PROGRAM G7_Palpage_Sommet_L
VAR_INPUT	SFCInit:BOOL;	END_VAR
VAR

	a1: LREAL;
	b1: LREAL;
	test_PalpSommet:BOOL;
END_VAR

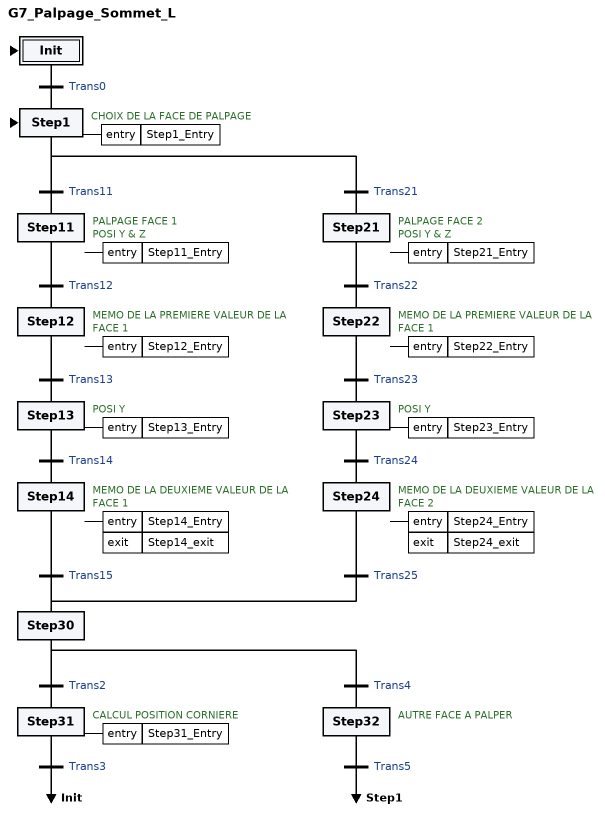
INITIAL_STEP Init:
END_STEP
TRANSITION FROM Init TO Step1
    := Trans0;
END_TRANSITION
// CHOIX DE LA FACE DE PALPAGE
STEP Step1:
    Step1_Entry(P1);  // entry action
END_STEP
TRANSITION FROM Step1 TO Step11
    := Trans11;
END_TRANSITION
// 																PALPAGE FACE 1
// POSI Y & Z
//
STEP Step11:
    Step11_Entry(P1);  // entry action
END_STEP
TRANSITION FROM Step11 TO Step12
    := Trans12;
END_TRANSITION
// MEMO DE LA PREMIERE VALEUR DE LA FACE 1
STEP Step12:
    Step12_Entry(P1);  // entry action
END_STEP
TRANSITION FROM Step12 TO Step13
    := Trans13;
END_TRANSITION
// POSI Y
STEP Step13:
    Step13_Entry(P1);  // entry action
END_STEP
TRANSITION FROM Step13 TO Step14
    := Trans14;
END_TRANSITION
// MEMO DE LA DEUXIEME VALEUR DE LA FACE 1
STEP Step14:
    Step14_Entry(P1);  // entry action
    Step14_exit(P0);  // exit action
END_STEP
TRANSITION FROM Step14 TO Step30
    := Trans15;
END_TRANSITION
TRANSITION FROM Step1 TO Step21
    := Trans21;
END_TRANSITION
// 																PALPAGE FACE 2
// POSI Y & Z
//
STEP Step21:
    Step21_Entry(P1);  // entry action
END_STEP
TRANSITION FROM Step21 TO Step22
    := Trans22;
END_TRANSITION
// MEMO DE LA PREMIERE VALEUR DE LA FACE 1
STEP Step22:
    Step22_Entry(P1);  // entry action
END_STEP
TRANSITION FROM Step22 TO Step23
    := Trans23;
END_TRANSITION
// POSI Y
STEP Step23:
    Step23_Entry(P1);  // entry action
END_STEP
TRANSITION FROM Step23 TO Step24
    := Trans24;
END_TRANSITION
// MEMO DE LA DEUXIEME VALEUR DE LA FACE 2
STEP Step24:
    Step24_Entry(P1);  // entry action
    Step24_exit(P0);  // exit action
END_STEP
TRANSITION FROM Step24 TO Step30
    := Trans25;
END_TRANSITION
STEP Step30:
END_STEP
TRANSITION FROM Step30 TO Step31
    := Trans2;
END_TRANSITION
TRANSITION FROM Step30 TO Step32
    := Trans4;
END_TRANSITION
// AUTRE FACE A PALPER
STEP Step32:
END_STEP
TRANSITION FROM Step32 TO Step1
    := Trans5;
END_TRANSITION
// 										CALCUL POSITION CORNIERE
//
//
STEP Step31:
    Step31_Entry(P1);  // entry action
END_STEP
TRANSITION FROM Step31 TO Init
    := Trans3;
END_TRANSITION

ACTION Step1_Entry:
CASE Face_Cible_Cycle OF	  
	1 : IF NOT Palpage_OK_Face_2 THEN
			Top_Palpage_Face_2 := TRUE;
			Top_Palpage_Face_1 := FALSE;
		ELSIF NOT Palpage_OK_Face_1 THEN
			Top_Palpage_Face_1 := TRUE;
			Top_Palpage_Face_2 := FALSE;
		ELSE
			Top_Palpage_Face_1 := FALSE;
			Top_Palpage_Face_2 := FALSE;
		END_IF;

	2,3 : 	IF NOT Palpage_OK_Face_1 THEN
			Top_Palpage_Face_1 := TRUE;
			Top_Palpage_Face_2 := FALSE;
		ELSIF NOT Palpage_OK_Face_2 THEN
			Top_Palpage_Face_2 := TRUE;
			Top_Palpage_Face_1 := FALSE;
		ELSE
			Top_Palpage_Face_1 := FALSE;
			Top_Palpage_Face_2 := FALSE;
		END_IF;
END_CASE;


IF Top_Palpage_Face_1 THEN
	 Face_Cible_Palpage := 1;
ELSIF  Top_Palpage_Face_2 THEN
	 Face_Cible_Palpage := 2;
ELSE
	Face_Cible_Palpage := 0;
END_IF;


IF Face_Cible_Palpage <> 0 THEN
	Face_Cible 		:= Face_Cible_Palpage;
	Face_En_Pos 	:= FALSE;
	Top_Face 		:= TRUE;
END_IF;
END_ACTION

ACTION Step11_Entry:
Pos_cible_Y_Laser := Offset_Y_Laser_REF + Hauteur_Aile - Ep_Ame - 5;
En_pos_Y_Laser :=FALSE;
Top_Y_Laser := TRUE;

Pos_cible_Z_Laser := Offset_Z_Laser_REF - Global_Divers.EP_Aile - 10;	//10 sécu arbitraire, à peut être adapter selon test
En_pos_Z_Laser :=FALSE;
Top_Z_Laser := TRUE;
END_ACTION

ACTION Step12_Entry:
Memo_Face_1_Y_1 := Hauteur_Aile - Ep_Ame - 5;
Memo_Face_1_Z_1 := Global_Divers.EP_Aile + Prog_Capacitance_Actual_Value_mm - 10;
END_ACTION

ACTION Step13_Entry:
Pos_cible_Y_Laser := Offset_Y_Laser_REF;
En_pos_Y_Laser :=FALSE;
Top_Y_Laser := TRUE;
END_ACTION

ACTION Step14_Entry:
Memo_Face_1_Y_2 := Ep_Ame;
Memo_Face_1_Z_2 := Global_Divers.EP_Aile + Prog_Capacitance_Actual_Value_mm - 10;
END_ACTION

ACTION Step14_exit:
Palpage_OK_Face_1:=true;
END_ACTION

ACTION Step21_Entry:
Pos_cible_Y_Laser := Offset_Y_Laser_OPP_REF - Largeur_Ame + Global_Divers.EP_Aile + 5;
En_pos_Y_Laser :=FALSE;
Top_Y_Laser := TRUE;

Pos_cible_Z_Laser := Offset_Z_Laser_OPP_REF - Ep_Ame - 10;
En_pos_Z_Laser :=FALSE;
Top_Z_Laser := TRUE;
END_ACTION

ACTION Step22_Entry:
Memo_Face_2_Y_1 := Largeur_Ame - Global_Divers.EP_Aile - 5;
Memo_Face_2_Z_1 := Ep_Ame + Prog_Capacitance_Actual_Value_mm - 10;
END_ACTION

ACTION Step23_Entry:
Pos_cible_Y_Laser := Offset_Y_Laser_OPP_REF;
En_pos_Y_Laser :=FALSE;
Top_Y_Laser := TRUE;
END_ACTION

ACTION Step24_Entry:
Memo_Face_2_Y_1 := Global_Divers.EP_Aile;
Memo_Face_2_Z_1 := Ep_Ame + Prog_Capacitance_Actual_Value_mm - 10;
END_ACTION

ACTION Step24_exit:
Palpage_OK_Face_2:=true;
END_ACTION

ACTION Step31_Entry:
(* Calcul a1 du coefficient Directeur de la Droite Coté Aile REF *)
a1 := (Memo_Face_1_Y_1 - Memo_Face_1_Y_2) / (Memo_Face_1_Z_1 / Memo_Face_1_Z_2);

(* Calcul de l'Ordonnée à l'Origine b1 de la Droite Coté Aile REF *)
b1 := Memo_Face_1_Y_1 - (a1 * Memo_Face_1_Z_1);


SHARK := SHARK;

Top_Palpage_Sommet:=false;
END_ACTION

TRANSITION Trans0:
(Auto OR test_PalpSommet)
AND (NOT Palpage_OK_Face_1 OR NOT Palpage_OK_Face_2)
AND Prog_Capacitance_Calibration_OK AND NOT Nv_ProcessID		
AND Top_Palpage_Sommet
END_TRANSITION

TRANSITION Trans11:
NOT Top_Face 				AND
Face_En_Pos 				AND
Face_Cible <> 0 				AND
Face_Cible = Face_En_Cours	AND

Top_Palpage_Face_1			AND
Face_En_Cours = 1
END_TRANSITION

TRANSITION Trans12:
En_pos_Y_Laser AND NOT Top_Y_Laser AND En_pos_Z_Laser AND NOT Top_Z_Laser
END_TRANSITION

TRANSITION Trans13:
step12.t>t#20ms
END_TRANSITION

TRANSITION Trans14:
En_pos_Y_Laser AND NOT Top_Y_Laser
END_TRANSITION

TRANSITION Trans15:
TRUE
END_TRANSITION

TRANSITION Trans2:
(Palpage_OK_Face_1 AND Palpage_OK_Face_2)
END_TRANSITION

TRANSITION Trans21:
NOT Top_Face 				AND
Face_En_Pos 				AND
Face_Cible <> 0 				AND
Face_Cible = Face_En_Cours	AND

Top_Palpage_Face_2			AND
Face_En_Cours = 2
END_TRANSITION

TRANSITION Trans22:
En_pos_Y_Laser AND NOT Top_Y_Laser AND En_pos_Z_Laser AND NOT Top_Z_Laser
END_TRANSITION

TRANSITION Trans23:
TRUE
END_TRANSITION

TRANSITION Trans24:
En_pos_Y_Laser AND NOT Top_Y_Laser
END_TRANSITION

TRANSITION Trans25:
TRUE
END_TRANSITION

TRANSITION Trans3:
NOT Top_Palpage_Sommet 
AND Palpage_OK_Face_1 
and Palpage_OK_Face_2
END_TRANSITION

TRANSITION Trans4:
(NOT Palpage_OK_Face_1 OR NOT Palpage_OK_Face_2)
END_TRANSITION

TRANSITION Trans5:
TRUE
END_TRANSITION

END_PROGRAM

(* stored: Version 1.1.0.1
   POU G7_Palpage_Sommet_L: Id {79df9942-df04-4b15-9230-d61f253b287b}, SpecialFunc None
   Action Step1_Entry: Id {0e2edc6f-315f-464d-b117-65620e2b1c8a}
   Action Step11_Entry: Id {d3e4a425-4f75-4489-ab57-2fd9e3ea4b31}
   Action Step12_Entry: Id {1a9c9888-7660-4a28-968f-965e7f79d8db}
   Action Step13_Entry: Id {87608582-0c6a-4296-9e6b-8a19c4719899}
   Action Step14_Entry: Id {42c18ed7-64e5-42eb-b781-a99e44c17d35}
   Action Step14_exit: Id {6cd4c35c-4470-4750-ac9a-bcadc656f321}
   Action Step21_Entry: Id {ae89a6af-92b1-4b55-a8c4-f4503c7fda92}
   Action Step22_Entry: Id {a69176f2-99f9-47d0-9c84-d9bf2b24368c}
   Action Step23_Entry: Id {91dac981-640f-4fc0-ad59-4055b62b771d}
   Action Step24_Entry: Id {a1635e56-47da-4a25-9fe5-7547e605c28f}
   Action Step24_exit: Id {51760de6-a85d-4f4c-90b9-7a83d918e0a1}
   Action Step31_Entry: Id {ca6bbbd1-dac4-4bb0-8155-620b7ec06320}
   Transition Trans0: Id {c3d12cc7-04f9-4bde-8a2d-8593d31a221c}
   Transition Trans11: Id {4b2b88a7-263f-4999-8453-23c5bb86f589}
   Transition Trans12: Id {dd96ba56-a463-4e8d-8bc1-db0be054d307}
   Transition Trans13: Id {0a503bde-9d7a-4d5e-8c20-4cf716968d74}
   Transition Trans14: Id {d46613e4-a492-434d-80a4-b37edf5a2690}
   Transition Trans15: Id {571755b3-da75-4ed7-b8e8-9c33b04d02f6}
   Transition Trans2: Id {22133bc6-87a4-49c1-9b48-fd6632a76d97}
   Transition Trans21: Id {961c6e79-3498-4ff5-9c7e-bf5244c7e419}
   Transition Trans22: Id {15be584b-9cf0-43d0-ab68-d8219ed8afb7}
   Transition Trans23: Id {874a2cf8-452e-45d7-81cc-fd2c96616461}
   Transition Trans24: Id {7388a26f-2a30-4ead-a7cb-6c21a53d0276}
   Transition Trans25: Id {479b1516-9e2f-4e68-8c5e-c777dfb4c7c6}
   Transition Trans3: Id {afe05620-b5de-4189-8241-76272c74888a}
   Transition Trans4: Id {a8b0fe86-2c25-4573-97d9-54fc8e6d3e38}
   Transition Trans5: Id {b162ef49-608c-43f3-8b07-8f91e84fe19e} *)
